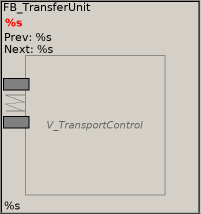
VISUALIZATION V_TransferUnit  // 201x214
VAR_IN_OUT
	{attribute 'VAR_IN_OUT_AS_POINTER'}
	fbFunction		: FB_TransferUnit;	
END_VAR
    Rectangle (0,0 200x214), colour toggle: fbFunction.Outputs.Drive_Run_12 OR fbFunction.Outputs.Drive_Run_21 OR fbFunction.Outputs.Drive_Run_34 OR fbFunction.Outputs.Drive_Run_43
    Rectangle (1,198 200x16), "%s", text variable: fbFunction.ConfigFunction.Zone[1].ZoneName
    Label (0,0 200x15), "FB_TransferUnit"
    Frame (25,55 140x140)
        shows V_TransportControl(TransportControl := fbFunction.fbTransportControl, ZoneData := fbFunction.ZoneData[1])
    Rectangle (2,15 196x16), "%s", tooltip "%s", text variable: fbFunction.FunctionData.ErrorData.Error.ErrorCode.Conv, invisible if: fbFunction.FunctionData.ErrorData.ErrorState = E_ErrorState.OPERATIONAL
        p4168582468: fbFunction.FunctionData.ErrorData.Error.ErrorParam
    Rectangle (3,116 26x12), tooltip "Lower lift sensor", colour toggle: fbFunction.HW_Inputs.Sensor_Pos_Down
    Rectangle (3,78 26x12), tooltip "Upper lift sensor", colour toggle: fbFunction.HW_Inputs.Sensor_Pos_Up
    Polyline (25,95) (6,95) (25,102) (6,104) (25,111) (6,111), colour toggle: fbFunction.HW_Outputs.Drive_Run_UpDown
    Rectangle (1,31 200x13), "Prev: %s", tooltip "FunctionInterface.in.ePrevFunctionNumber", text variable: fbFunction.FunctionInterface.In.ePrevFunctionNumber
    Rectangle (1,43 200x13), "Next: %s", tooltip "FunctionInterface.in.eNextFunctionNumber", text variable: fbFunction.FunctionInterface.In.eNextFunctionNumber
END_VISUALIZATION

(* stored: Version 1.1.0.1, ProductVersion 3.1.4024.9
   Visu V_TransferUnit: Id {a4aaaa59-827b-45d8-9d47-416931efd5d5} *)
